FUNCTION_BLOCK STRINGTEST (* Test String Assignments *)
  (* Standard: 61499-2 *)
  (* Version 0.0, 2003-11-14, JHC, Rockwell Automation *)
  (* Compiler header: package fb.rt.test; *)
  (* Compiler Java IBM Jikes 1.06 *)
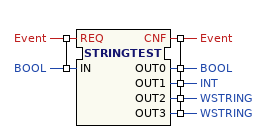
  EVENT_INPUT
    REQ WITH IN; (* Normal Execution Request *)
  END_EVENT
  EVENT_OUTPUT
    CNF WITH OUT0, OUT1, OUT2, OUT3; (* Execution Confirmation *)
  END_EVENT
  VAR_INPUT
    IN : BOOL; (* Input *)
  END_VAR
  VAR_OUTPUT
    OUT0 : BOOL; (* Boolean output *)
    OUT1 : INT; (* Integer output *)
    OUT2 : WSTRING; (* String output *)
    OUT3 : WSTRING; (* String output *)
  END_VAR
  ALGORITHM REQ IN ST:
OUT0:=IN;
IF IN THEN
OUT1:=1;
OUT2 := "Input is  $"true$"";
OUT3 := "Input is  $'true'";
ELSE
OUT1:=0;
OUT2 := "Input is $"false$"";
OUT3 := "Input is $'false$'";
END_IF
CNF.serviceEvent(this);
  END_ALGORITHM
END_FUNCTION_BLOCK
